FUNCTION_BLOCK FB_RV_St
VAR_IN_OUT
END_VAR
VAR_INPUT
END_VAR
VAR_OUTPUT
	{attribute 'OPC.UA.DA' := '1'}Zustand					: ST_RV_Zustand;
	{attribute 'OPC.UA.DA' := '1'}Parameter				: ST_RV_Parameter;	
END_VAR
VAR
	Zustandscheck			: FB_RV_St_Zustandscheck;
END_VAR

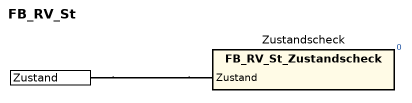
Zustandscheck(Zustand := Zustand); // FB_RV_St_Zustandscheck

END_FUNCTION_BLOCK

(* stored: Version 1.1.0.1, ProductVersion 3.1.4024.9
   POU FB_RV_St: Id {74fde8ad-06fc-43f7-bc6e-70e6961ea171}, SpecialFunc None *)
